{attribute addProperty BoxType "EL3403-0000-0017"}
{attribute addProperty Id "Missing_zero_crossing_AAT %I*BOOL814Missing_zero_crossing_BAT %I*BOOL815Missing_zero_crossing_CAT %I*BOOL816Phase_sequence_errorAT %I*BOOL819Sync_ErrorAT %I*BOOL8114"}
{attribute addProperty CRC "3426899727"}
{attribute addProperty SizeInBites "40"}
{attribute addProperty SizeInBytes "5"}
TYPE PM_Status_data_CC42570F :
STRUCT
	{attribute addProperty Name "Missing_zero_crossing_A"}
	Missing_zero_crossing_A AT %I* : BOOL;
	{attribute addProperty Name "Missing_zero_crossing_B"}
	Missing_zero_crossing_B AT %I* : BOOL;
	{attribute addProperty Name "Missing_zero_crossing_C"}
	Missing_zero_crossing_C AT %I* : BOOL;
	{attribute addProperty Name "Phase_sequence_error"}
	Phase_sequence_error AT %I* : BOOL;
	{attribute addProperty Name "Sync_Error"}
	Sync_Error AT %I* : BOOL;
END_STRUCT
END_TYPE

(* stored: Version 1.2.0.0, ProductVersion 3.1.4024.9
   DUT PM_Status_data_CC42570F: Id {6df6f125-1737-4712-bdbf-f0188626aa5c} *)
